// TIA Portal V20 export
FUNCTION_BLOCK "zFNet_10Child"   // FB218, LAD
// stored: MemoryReserve 100, Namespace CITI_Logic, SetENOAutomatically false
   VAR_INPUT
      IN_NumberOf_FN_Retries : Int;   // Number of Timers to Retry the Connection to FNet
      IN_Component_Quantity : Int;   // Number of Child Components
      IN_FN_Response_FLT_Time : DInt;
      IN_OEM_Data : "CITI_Logic.FlexNet_Data";
   END_VAR
   VAR_OUTPUT
      FN_Data : "CITI_Logic.FlexNet_Data";
      FlexNet_White_Light : Bool;
      FlexNet_Green_Light : Bool;
      FlexNet_Buzzer : Bool;
      FlexNet_No_Response_Count : Int;
      FlexNet_DataReceivedByHost : Bool;
      FlexNet_Last_ResponseTime : DInt;
   END_VAR
   VAR
      FN_Dry_Cycle_Block : Bool;
      FN_OneShot : Array[1..32] of Bool;
      Clock_Data : DTL;   // Clock Data used for FlexNet Time Stamp
      System_Time_Tick : Time;   // System Time Tick
      Present_Time_Tick : Int;   // Present Time Tick
      Previous_Time_Tick : Int;   // Previous Time Tick
      Difference_Time_Tick : Int;   // Difference between Present and Previous Tick
      Difference_Time_DInt : DInt;   // Difference in Time
      TimerForFN_DataReady : DInt;   // FlexNet Data Ready Delay
      TimerForFN_Response_Test : DInt;   // FlexNet Response Test
      TimerFN_DataReady_Retry : DInt;   // FlexNet Data Ready Retry Delay
      TimerFN_BuzzerOn : DInt;   // FlexNet No Response Buzzer
      FN_PUNDataRdy_Dly : Bool;   // Start Data Ready Timer
      FN_DataReady_Failed_Retry : Bool;
      FlasherOn : Bool;   // Flasher for StackLights
      FN_NumberOf_Retries : Int;
      FN_Num_Of_Retry_Cnt_HMI : Int;
      FlexNet_Response_FLT_CNT : Int;
      TimerForFlasher : DInt;
      FN_Data_Recd_Delay : Bool;
      Timer_HQ_Delay : DInt;   // FlexNet No Response Buzzer
      Timer_GreenLight_Delay : DInt;   // FlexNet No Response Buzzer
      FN_Num_Of_Retries_CNT : Int;
   END_VAR
   VAR DB_SPECIFIC
      FlexNet_Part_Passed { ExternalAccessible := 'False'; ExternalVisible := 'False'; ExternalWritable := 'False'} : Bool;   // Calculated Part Passed
      FlexNet_Part_Failed { ExternalAccessible := 'False'; ExternalVisible := 'False'; ExternalWritable := 'False'} : Bool;   // Calculated Part Failed
   END_VAR
   VAR
      FlexNet_PassFail_Valid { ExternalAccessible := 'False'; ExternalVisible := 'False'; ExternalWritable := 'False'} : Bool;   // Calculated Valid Part Fail/Pass Data
      ON { ExternalAccessible := 'False'; ExternalVisible := 'False'; ExternalWritable := 'False'} : Bool;   // On
      OFF { ExternalAccessible := 'False'; ExternalVisible := 'False'; ExternalWritable := 'False'} : Bool;   // Off
      ReadClock_Rslt { ExternalAccessible := 'False'; ExternalVisible := 'False'; ExternalWritable := 'False'} : Int;
   END_VAR
   VAR_TEMP   // added for the SCL form of the ladder/FBD networks
      _w1 : Bool;
      _w2 : Bool;
      _w3 : Bool;
      _w4 : Bool;
   END_VAR
BEGIN

REGION Network 1: Always ON and Always OFF Setup
   // Generate local "Always ON" and "Always OFF" conditions
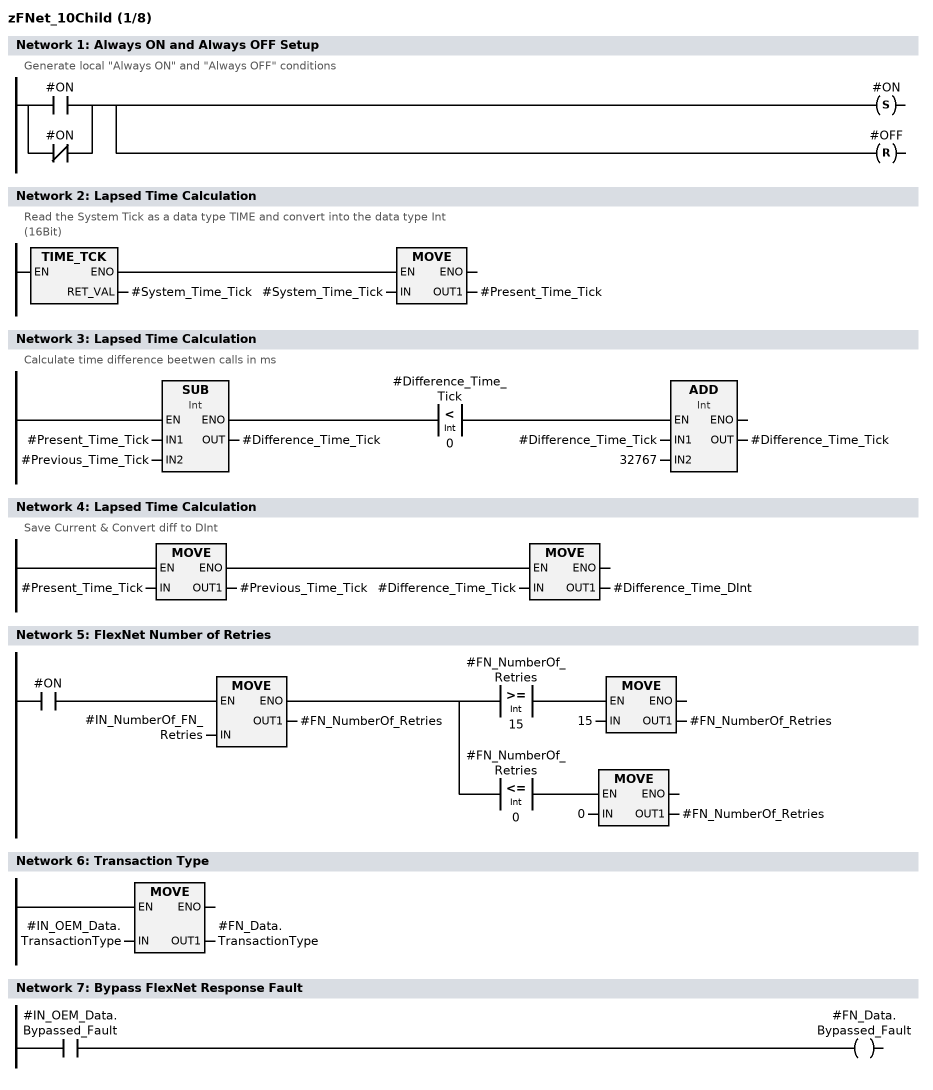
   RUNG wire#powerrail
      Contact( #ON )
      wire#w1
      S_Coil( #ON )
   END_RUNG
   RUNG wire#powerrail
      I_Contact( #ON )
   END_RUNG wire#w1
   RUNG wire#w1
      R_Coil( #OFF )
   END_RUNG
   // the same network as SCL:
   #_w1 := #ON OR NOT #ON;
   IF #_w1 THEN
       #ON := TRUE;
       #OFF := FALSE;
   END_IF;
END_REGION

REGION Network 2: Lapsed Time Calculation
   // Read the System Tick as a data type TIME and convert into the data type Int 
   // (16Bit)
   RUNG wire#powerrail
      TIME_TCK(RET_VAL => #System_Time_Tick)
      { S7_GenerateENO := "TRUE" } Move(in := #System_Time_Tick, out1 => #Present_Time_Tick)
   END_RUNG
   // the same network as SCL:
   #System_Time_Tick := TIME_TCK(ENO => #_w1);
   IF #_w1 THEN #Present_Time_Tick := #System_Time_Tick; END_IF;
END_REGION

REGION Network 3: Lapsed Time Calculation
   // Calculate time difference beetwen calls in ms
   RUNG wire#powerrail
      { S7_Templates := "SrcType := Int"; S7_GenerateENO := "TRUE" } Sub(in1 := #Present_Time_Tick, in2 := #Previous_Time_Tick, out => #Difference_Time_Tick)
      { S7_Templates := "SrcType := Int" } LT_Contact(in1 := #Difference_Time_Tick, in2 := 0)
      { S7_Templates := "SrcType := Int"; S7_GenerateENO := "TRUE" } Add(in1 := #Difference_Time_Tick, in2 := 32767, out => #Difference_Time_Tick)
   END_RUNG
   // the same network as SCL:
   // ENO of a box is taken as its EN; it also drops when the box reports an error
   #Difference_Time_Tick := #Present_Time_Tick - #Previous_Time_Tick;
   IF #Difference_Time_Tick < 0 THEN #Difference_Time_Tick := #Difference_Time_Tick + 32767; END_IF;
END_REGION

REGION Network 4: Lapsed Time Calculation
   // Save Current & Convert diff to DInt
   RUNG wire#powerrail
      { S7_GenerateENO := "TRUE" } Move(in := #Present_Time_Tick, out1 => #Previous_Time_Tick)
      { S7_GenerateENO := "TRUE" } Move(in := #Difference_Time_Tick, out1 => #Difference_Time_DInt)
   END_RUNG
   // the same network as SCL:
   // ENO of a box is taken as its EN; it also drops when the box reports an error
   #Previous_Time_Tick := #Present_Time_Tick;
   #Difference_Time_DInt := #Difference_Time_Tick;
END_REGION

REGION Network 5: FlexNet Number of Retries
   RUNG wire#powerrail
      Contact( #ON )
      { S7_GenerateENO := "TRUE" } Move(in := #IN_NumberOf_FN_Retries, out1 => #FN_NumberOf_Retries)
      wire#w1
      { S7_Templates := "SrcType := Int" } GE_Contact(in1 := #FN_NumberOf_Retries, in2 := 15)
      { S7_GenerateENO := "TRUE" } Move(in := 15, out1 => #FN_NumberOf_Retries)
   END_RUNG
   RUNG wire#w1
      { S7_Templates := "SrcType := Int" } LE_Contact(in1 := #FN_NumberOf_Retries, in2 := 0)
      { S7_GenerateENO := "TRUE" } Move(in := 0, out1 => #FN_NumberOf_Retries)
   END_RUNG
   // the same network as SCL:
   // ENO of a box is taken as its EN; it also drops when the box reports an error
   IF #ON THEN #FN_NumberOf_Retries := #IN_NumberOf_FN_Retries; END_IF;
   IF #ON AND (#FN_NumberOf_Retries >= 15) THEN #FN_NumberOf_Retries := 15; END_IF;
   IF #ON AND (#FN_NumberOf_Retries <= 0) THEN #FN_NumberOf_Retries := 0; END_IF;
END_REGION

REGION Network 6: Transaction Type
   RUNG wire#powerrail
      { S7_GenerateENO := "TRUE" } Move(in := #IN_OEM_Data.TransactionType, out1 => #FN_Data.TransactionType)
   END_RUNG
   // the same network as SCL:
   #FN_Data.TransactionType := #IN_OEM_Data.TransactionType;
END_REGION

REGION Network 7: Bypass FlexNet Response Fault
   RUNG wire#powerrail
      Contact( #IN_OEM_Data.Bypassed_Fault )
      Coil( #FN_Data.Bypassed_Fault )
   END_RUNG
   // the same network as SCL:
   #FN_Data.Bypassed_Fault := #IN_OEM_Data.Bypassed_Fault;
END_REGION

REGION Network 8: Data Reset Input
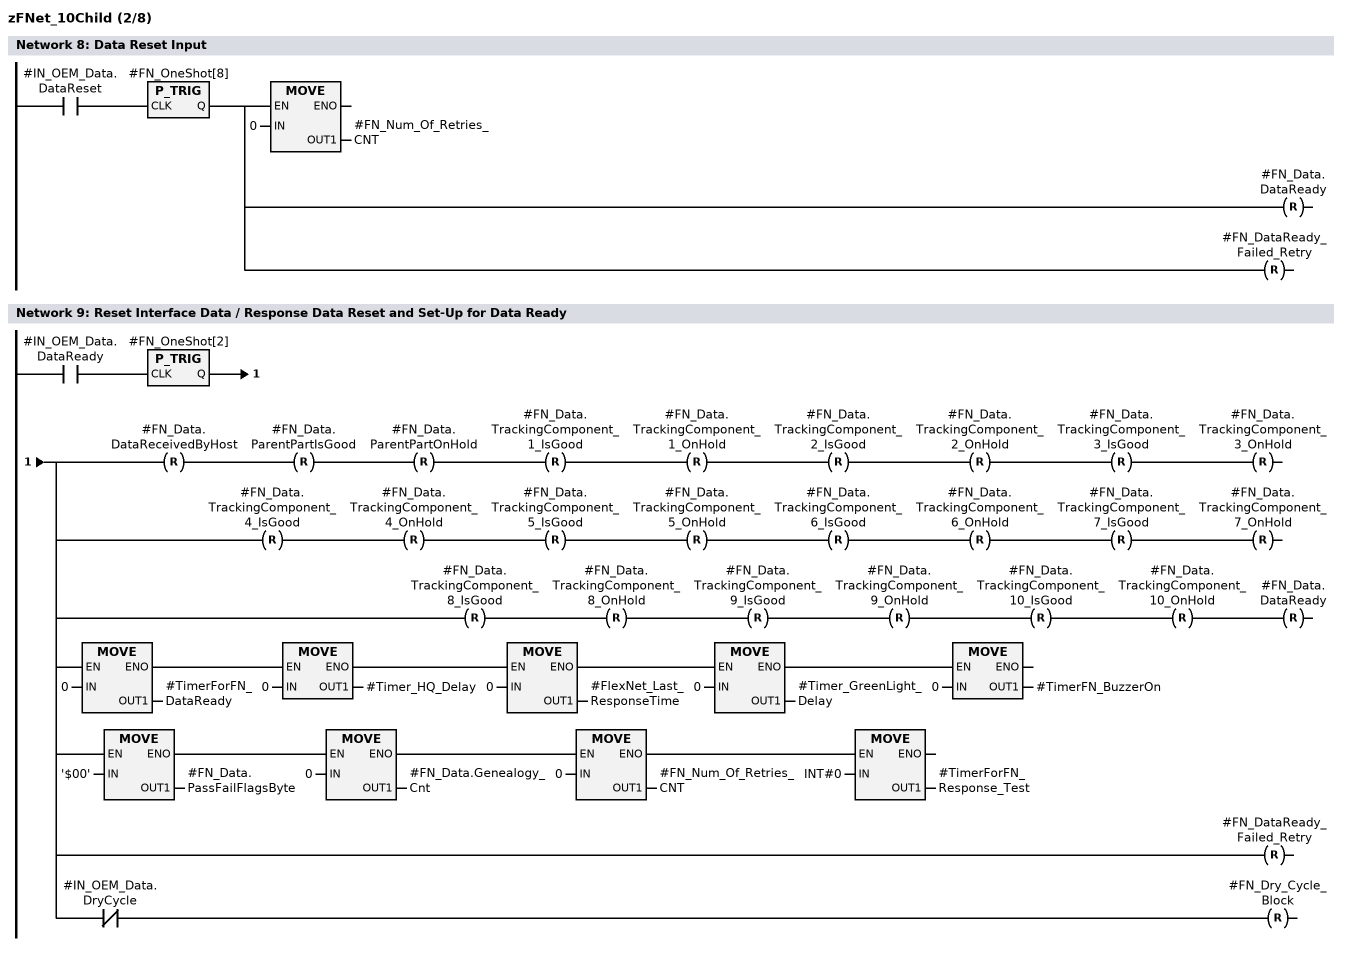
   RUNG wire#powerrail
      Contact( #IN_OEM_Data.DataReset )
      P_Trig( #FN_OneShot[8] )
      wire#w1
      { S7_GenerateENO := "TRUE" } Move(in := 0, out1 => #FN_Num_Of_Retries_CNT)
   END_RUNG
   RUNG wire#w1
      R_Coil( #FN_Data.DataReady )
   END_RUNG
   RUNG wire#w1
      R_Coil( #FN_DataReady_Failed_Retry )
   END_RUNG
   // the same network as SCL:
   #_w1 := #IN_OEM_Data.DataReset AND NOT #FN_OneShot[8];   // rising edge
   #FN_OneShot[8] := #IN_OEM_Data.DataReset;
   IF #_w1 THEN
       #FN_Num_Of_Retries_CNT := 0;
       #FN_Data.DataReady := FALSE;
       #FN_DataReady_Failed_Retry := FALSE;
   END_IF;
END_REGION

REGION Network 9: Reset Interface Data / Response Data Reset and Set-Up for Data Ready
   RUNG wire#powerrail
      Contact( #IN_OEM_Data.DataReady )
      P_Trig( #FN_OneShot[2] )
      wire#w1
      R_Coil( #FN_Data.DataReceivedByHost )
      R_Coil( #FN_Data.ParentPartIsGood )
      R_Coil( #FN_Data.ParentPartOnHold )
      R_Coil( #FN_Data.TrackingComponent_1_IsGood )
      R_Coil( #FN_Data.TrackingComponent_1_OnHold )
      R_Coil( #FN_Data.TrackingComponent_2_IsGood )
      R_Coil( #FN_Data.TrackingComponent_2_OnHold )
      R_Coil( #FN_Data.TrackingComponent_3_IsGood )
      R_Coil( #FN_Data.TrackingComponent_3_OnHold )
   END_RUNG
   RUNG wire#w1
      R_Coil( #FN_Data.TrackingComponent_4_IsGood )
      R_Coil( #FN_Data.TrackingComponent_4_OnHold )
      R_Coil( #FN_Data.TrackingComponent_5_IsGood )
      R_Coil( #FN_Data.TrackingComponent_5_OnHold )
      R_Coil( #FN_Data.TrackingComponent_6_IsGood )
      R_Coil( #FN_Data.TrackingComponent_6_OnHold )
      R_Coil( #FN_Data.TrackingComponent_7_IsGood )
      R_Coil( #FN_Data.TrackingComponent_7_OnHold )
   END_RUNG
   RUNG wire#w1
      R_Coil( #FN_Data.TrackingComponent_8_IsGood )
      R_Coil( #FN_Data.TrackingComponent_8_OnHold )
      R_Coil( #FN_Data.TrackingComponent_9_IsGood )
      R_Coil( #FN_Data.TrackingComponent_9_OnHold )
      R_Coil( #FN_Data.TrackingComponent_10_IsGood )
      R_Coil( #FN_Data.TrackingComponent_10_OnHold )
      R_Coil( #FN_Data.DataReady )
   END_RUNG
   RUNG wire#w1
      Move(in := 0, out1 => #TimerForFN_DataReady)
      Move(in := 0, out1 => #Timer_HQ_Delay)
      Move(in := 0, out1 => #FlexNet_Last_ResponseTime)
      Move(in := 0, out1 => #Timer_GreenLight_Delay)
      { S7_GenerateENO := "TRUE" } Move(in := 0, out1 => #TimerFN_BuzzerOn)
   END_RUNG
   RUNG wire#w1
      { S7_GenerateENO := "TRUE" } Move(in := '$00', out1 => #FN_Data.PassFailFlagsByte)
      Move(in := 0, out1 => #FN_Data.Genealogy_Cnt)
      { S7_GenerateENO := "TRUE" } Move(in := 0, out1 => #FN_Num_Of_Retries_CNT)
      { S7_GenerateENO := "TRUE" } Move(in := INT#0, out1 => #TimerForFN_Response_Test)
   END_RUNG
   RUNG wire#w1
      R_Coil( #FN_DataReady_Failed_Retry )
   END_RUNG
   RUNG wire#w1
      I_Contact( #IN_OEM_Data.DryCycle )
      R_Coil( #FN_Dry_Cycle_Block )
   END_RUNG
   // the same network as SCL:
   // ENO of a box is taken as its EN; it also drops when the box reports an error
   #_w1 := #IN_OEM_Data.DataReady AND NOT #FN_OneShot[2];   // rising edge
   #FN_OneShot[2] := #IN_OEM_Data.DataReady;
   IF #_w1 THEN
       #FN_Data.DataReceivedByHost := FALSE;
       #FN_Data.ParentPartIsGood := FALSE;
       #FN_Data.ParentPartOnHold := FALSE;
       #FN_Data.TrackingComponent_1_IsGood := FALSE;
       #FN_Data.TrackingComponent_1_OnHold := FALSE;
       #FN_Data.TrackingComponent_2_IsGood := FALSE;
       #FN_Data.TrackingComponent_2_OnHold := FALSE;
       #FN_Data.TrackingComponent_3_IsGood := FALSE;
       #FN_Data.TrackingComponent_3_OnHold := FALSE;
       #FN_Data.TrackingComponent_4_IsGood := FALSE;
       #FN_Data.TrackingComponent_4_OnHold := FALSE;
       #FN_Data.TrackingComponent_5_IsGood := FALSE;
       #FN_Data.TrackingComponent_5_OnHold := FALSE;
       #FN_Data.TrackingComponent_6_IsGood := FALSE;
       #FN_Data.TrackingComponent_6_OnHold := FALSE;
       #FN_Data.TrackingComponent_7_IsGood := FALSE;
       #FN_Data.TrackingComponent_7_OnHold := FALSE;
       #FN_Data.TrackingComponent_8_IsGood := FALSE;
       #FN_Data.TrackingComponent_8_OnHold := FALSE;
       #FN_Data.TrackingComponent_9_IsGood := FALSE;
       #FN_Data.TrackingComponent_9_OnHold := FALSE;
       #FN_Data.TrackingComponent_10_IsGood := FALSE;
       #FN_Data.TrackingComponent_10_OnHold := FALSE;
       #FN_Data.DataReady := FALSE;
       #TimerForFN_DataReady := 0;
       #Timer_HQ_Delay := 0;
       #FlexNet_Last_ResponseTime := 0;
       #Timer_GreenLight_Delay := 0;
       #TimerFN_BuzzerOn := 0;
       #FN_Data.PassFailFlagsByte := '$00';
       #FN_Data.Genealogy_Cnt := 0;
       #FN_Num_Of_Retries_CNT := 0;
       #TimerForFN_Response_Test := INT#0;
       #FN_DataReady_Failed_Retry := FALSE;
   END_IF;
   IF #_w1 AND NOT #IN_OEM_Data.DryCycle THEN #FN_Dry_Cycle_Block := FALSE; END_IF;
END_REGION

REGION Network 10: Test Part Failed or Passed signals Using the Transaction Byte to enable certain test parameters
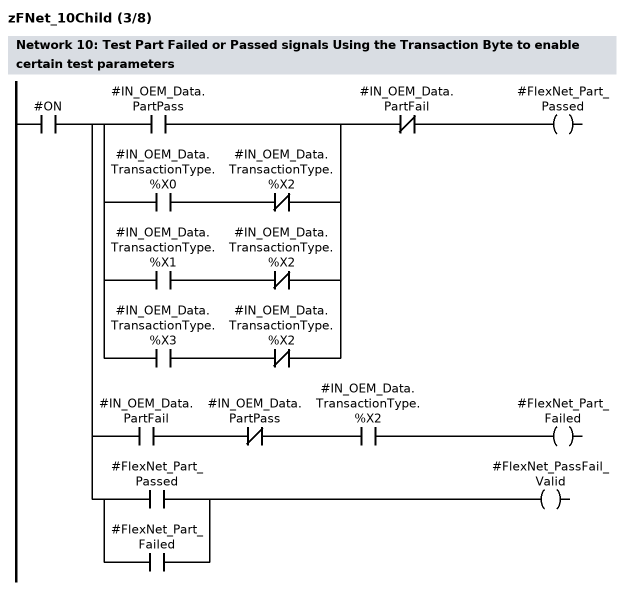
   RUNG wire#powerrail
      Contact( #ON )
      wire#w1
      Contact( #IN_OEM_Data.PartPass )
      wire#w2
      I_Contact( #IN_OEM_Data.PartFail )
      Coil( #FlexNet_Part_Passed )
   END_RUNG
   RUNG wire#w1
      Contact( #IN_OEM_Data.TransactionType.%X0 )
      I_Contact( #IN_OEM_Data.TransactionType.%X2 )
   END_RUNG wire#w2
   RUNG wire#w1
      Contact( #IN_OEM_Data.TransactionType.%X1 )
      I_Contact( #IN_OEM_Data.TransactionType.%X2 )
   END_RUNG wire#w2
   RUNG wire#w1
      Contact( #IN_OEM_Data.TransactionType.%X3 )
      I_Contact( #IN_OEM_Data.TransactionType.%X2 )
   END_RUNG wire#w2
   RUNG wire#w1
      Contact( #IN_OEM_Data.PartFail )
      I_Contact( #IN_OEM_Data.PartPass )
      Contact( #IN_OEM_Data.TransactionType.%X2 )
      Coil( #FlexNet_Part_Failed )
   END_RUNG
   RUNG wire#w1
      Contact( #FlexNet_Part_Passed )
      wire#w3
      Coil( #FlexNet_PassFail_Valid )
   END_RUNG
   RUNG wire#w1
      Contact( #FlexNet_Part_Failed )
   END_RUNG wire#w3
   // the same network as SCL:
   #FlexNet_Part_Passed := #ON AND (#IN_OEM_Data.PartPass OR (#IN_OEM_Data.TransactionType.%X0 AND NOT #IN_OEM_Data.TransactionType.%X2) OR (#IN_OEM_Data.TransactionType.%X1 AND NOT #IN_OEM_Data.TransactionType.%X2) OR (#IN_OEM_Data.TransactionType.%X3 AND NOT #IN_OEM_Data.TransactionType.%X2)) AND NOT #IN_OEM_Data.PartFail;
   #FlexNet_Part_Failed := #ON AND #IN_OEM_Data.PartFail AND NOT #IN_OEM_Data.PartPass AND #IN_OEM_Data.TransactionType.%X2;
   #FlexNet_PassFail_Valid := #ON AND (#FlexNet_Part_Passed OR #FlexNet_Part_Failed);
END_REGION

REGION Network 11: Copy PUN Data, Tracking ID/Attribute, Clock Data, Part Pass/Fail Data into FlexNet Registers
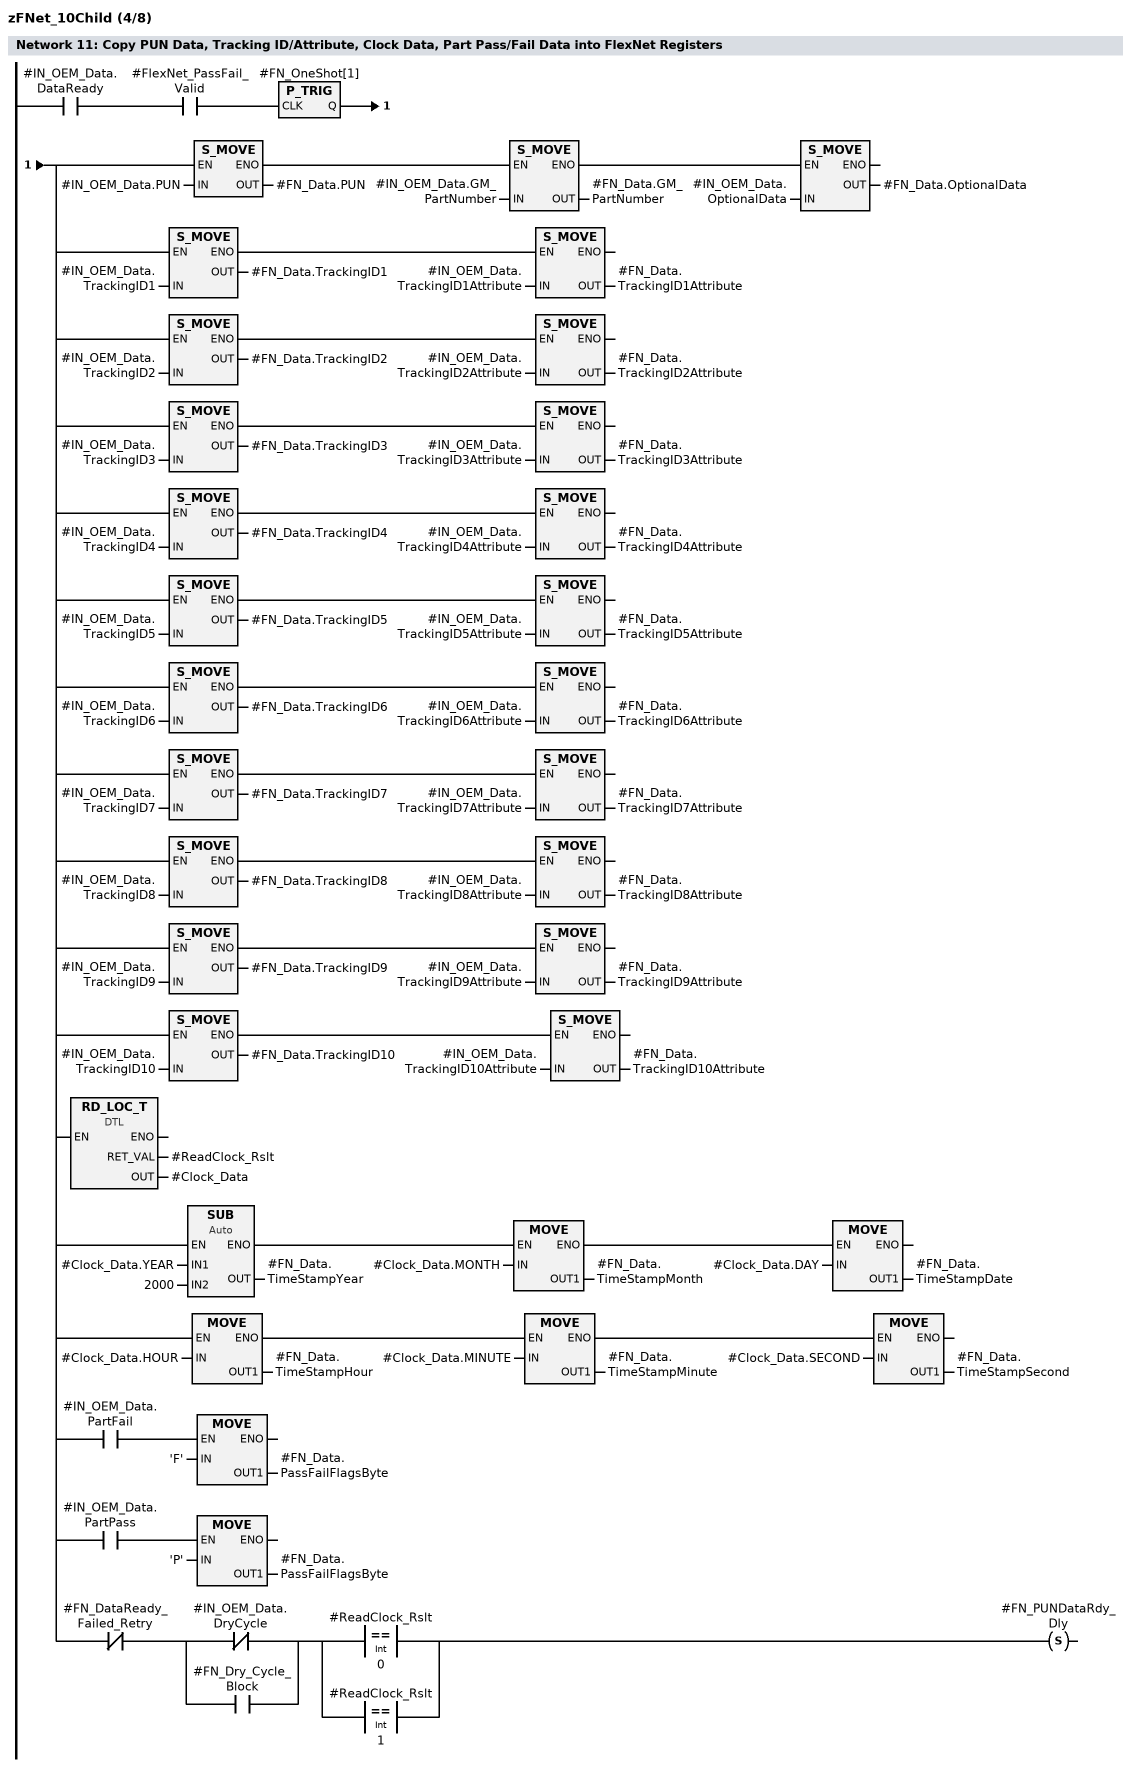
   RUNG wire#powerrail
      Contact( #IN_OEM_Data.DataReady )
      Contact( #FlexNet_PassFail_Valid )
      P_Trig( #FN_OneShot[1] )
      wire#w1
      S_Move(in := #IN_OEM_Data.PUN, out => #FN_Data.PUN)
      S_Move(in := #IN_OEM_Data.GM_PartNumber, out => #FN_Data.GM_PartNumber)
      S_Move(in := #IN_OEM_Data.OptionalData, out => #FN_Data.OptionalData)
   END_RUNG
   RUNG wire#w1
      S_Move(in := #IN_OEM_Data.TrackingID1, out => #FN_Data.TrackingID1)
      S_Move(in := #IN_OEM_Data.TrackingID1Attribute, out => #FN_Data.TrackingID1Attribute)
   END_RUNG
   RUNG wire#w1
      S_Move(in := #IN_OEM_Data.TrackingID2, out => #FN_Data.TrackingID2)
      S_Move(in := #IN_OEM_Data.TrackingID2Attribute, out => #FN_Data.TrackingID2Attribute)
   END_RUNG
   RUNG wire#w1
      S_Move(in := #IN_OEM_Data.TrackingID3, out => #FN_Data.TrackingID3)
      S_Move(in := #IN_OEM_Data.TrackingID3Attribute, out => #FN_Data.TrackingID3Attribute)
   END_RUNG
   RUNG wire#w1
      S_Move(in := #IN_OEM_Data.TrackingID4, out => #FN_Data.TrackingID4)
      S_Move(in := #IN_OEM_Data.TrackingID4Attribute, out => #FN_Data.TrackingID4Attribute)
   END_RUNG
   RUNG wire#w1
      S_Move(in := #IN_OEM_Data.TrackingID5, out => #FN_Data.TrackingID5)
      S_Move(in := #IN_OEM_Data.TrackingID5Attribute, out => #FN_Data.TrackingID5Attribute)
   END_RUNG
   RUNG wire#w1
      S_Move(in := #IN_OEM_Data.TrackingID6, out => #FN_Data.TrackingID6)
      S_Move(in := #IN_OEM_Data.TrackingID6Attribute, out => #FN_Data.TrackingID6Attribute)
   END_RUNG
   RUNG wire#w1
      S_Move(in := #IN_OEM_Data.TrackingID7, out => #FN_Data.TrackingID7)
      S_Move(in := #IN_OEM_Data.TrackingID7Attribute, out => #FN_Data.TrackingID7Attribute)
   END_RUNG
   RUNG wire#w1
      S_Move(in := #IN_OEM_Data.TrackingID8, out => #FN_Data.TrackingID8)
      S_Move(in := #IN_OEM_Data.TrackingID8Attribute, out => #FN_Data.TrackingID8Attribute)
   END_RUNG
   RUNG wire#w1
      S_Move(in := #IN_OEM_Data.TrackingID9, out => #FN_Data.TrackingID9)
      S_Move(in := #IN_OEM_Data.TrackingID9Attribute, out => #FN_Data.TrackingID9Attribute)
   END_RUNG
   RUNG wire#w1
      S_Move(in := #IN_OEM_Data.TrackingID10, out => #FN_Data.TrackingID10)
      S_Move(in := #IN_OEM_Data.TrackingID10Attribute, out => #FN_Data.TrackingID10Attribute)
   END_RUNG
   RUNG wire#w1
      { S7_Templates := "date_type := DTL" } RD_LOC_T(RET_VAL => #ReadClock_Rslt, OUT => #Clock_Data)
   END_RUNG
   RUNG wire#w1
      Sub(in1 := #Clock_Data.YEAR, in2 := 2000, out => #FN_Data.TimeStampYear)
      Move(in := #Clock_Data.MONTH, out1 => #FN_Data.TimeStampMonth)
      Move(in := #Clock_Data.DAY, out1 => #FN_Data.TimeStampDate)
   END_RUNG
   RUNG wire#w1
      Move(in := #Clock_Data.HOUR, out1 => #FN_Data.TimeStampHour)
      Move(in := #Clock_Data.MINUTE, out1 => #FN_Data.TimeStampMinute)
      Move(in := #Clock_Data.SECOND, out1 => #FN_Data.TimeStampSecond)
   END_RUNG
   RUNG wire#w1
      Contact( #IN_OEM_Data.PartFail )
      Move(in := 'F', out1 => #FN_Data.PassFailFlagsByte)
   END_RUNG
   RUNG wire#w1
      Contact( #IN_OEM_Data.PartPass )
      Move(in := 'P', out1 => #FN_Data.PassFailFlagsByte)
   END_RUNG
   RUNG wire#w1
      I_Contact( #FN_DataReady_Failed_Retry )
      wire#w2
      I_Contact( #IN_OEM_Data.DryCycle )
      wire#w3
      { S7_Templates := "SrcType := Int" } EQ_Contact(in1 := #ReadClock_Rslt, in2 := 0)
      wire#w4
      S_Coil( #FN_PUNDataRdy_Dly )
   END_RUNG
   RUNG wire#w2
      Contact( #FN_Dry_Cycle_Block )
   END_RUNG wire#w3
   RUNG wire#w3
      { S7_Templates := "SrcType := Int" } EQ_Contact(in1 := #ReadClock_Rslt, in2 := 1)
   END_RUNG wire#w4
   // the same network as SCL:
   #_w1 := #IN_OEM_Data.DataReady AND #FlexNet_PassFail_Valid;
   #_w2 := #_w1 AND NOT #FN_OneShot[1];   // rising edge
   #FN_OneShot[1] := #_w1;
   IF #_w2 THEN
       #FN_Data.PUN := #IN_OEM_Data.PUN;
       #FN_Data.GM_PartNumber := #IN_OEM_Data.GM_PartNumber;
       #FN_Data.OptionalData := #IN_OEM_Data.OptionalData;
       #FN_Data.TrackingID1 := #IN_OEM_Data.TrackingID1;
       #FN_Data.TrackingID1Attribute := #IN_OEM_Data.TrackingID1Attribute;
       #FN_Data.TrackingID2 := #IN_OEM_Data.TrackingID2;
       #FN_Data.TrackingID2Attribute := #IN_OEM_Data.TrackingID2Attribute;
       #FN_Data.TrackingID3 := #IN_OEM_Data.TrackingID3;
       #FN_Data.TrackingID3Attribute := #IN_OEM_Data.TrackingID3Attribute;
       #FN_Data.TrackingID4 := #IN_OEM_Data.TrackingID4;
       #FN_Data.TrackingID4Attribute := #IN_OEM_Data.TrackingID4Attribute;
       #FN_Data.TrackingID5 := #IN_OEM_Data.TrackingID5;
       #FN_Data.TrackingID5Attribute := #IN_OEM_Data.TrackingID5Attribute;
       #FN_Data.TrackingID6 := #IN_OEM_Data.TrackingID6;
       #FN_Data.TrackingID6Attribute := #IN_OEM_Data.TrackingID6Attribute;
       #FN_Data.TrackingID7 := #IN_OEM_Data.TrackingID7;
       #FN_Data.TrackingID7Attribute := #IN_OEM_Data.TrackingID7Attribute;
       #FN_Data.TrackingID8 := #IN_OEM_Data.TrackingID8;
       #FN_Data.TrackingID8Attribute := #IN_OEM_Data.TrackingID8Attribute;
       #FN_Data.TrackingID9 := #IN_OEM_Data.TrackingID9;
       #FN_Data.TrackingID9Attribute := #IN_OEM_Data.TrackingID9Attribute;
       #FN_Data.TrackingID10 := #IN_OEM_Data.TrackingID10;
       #FN_Data.TrackingID10Attribute := #IN_OEM_Data.TrackingID10Attribute;
       #ReadClock_Rslt := RD_LOC_T(OUT => #Clock_Data);
       #FN_Data.TimeStampYear := #Clock_Data.YEAR - 2000;
       #FN_Data.TimeStampMonth := #Clock_Data.MONTH;
       #FN_Data.TimeStampDate := #Clock_Data.DAY;
       #FN_Data.TimeStampHour := #Clock_Data.HOUR;
       #FN_Data.TimeStampMinute := #Clock_Data.MINUTE;
       #FN_Data.TimeStampSecond := #Clock_Data.SECOND;
   END_IF;
   IF #_w2 AND #IN_OEM_Data.PartFail THEN #FN_Data.PassFailFlagsByte := 'F'; END_IF;
   IF #_w2 AND #IN_OEM_Data.PartPass THEN #FN_Data.PassFailFlagsByte := 'P'; END_IF;
   IF #_w2 AND NOT #FN_DataReady_Failed_Retry AND (NOT #IN_OEM_Data.DryCycle OR #FN_Dry_Cycle_Block) AND ((#ReadClock_Rslt = 0) OR (#ReadClock_Rslt = 1)) THEN
       #FN_PUNDataRdy_Dly := TRUE;
   END_IF;
END_REGION

REGION Network 12: Turn On FlexNet DataReady. Reset PUN Data Ready Delay and Failed Retry Data Ready
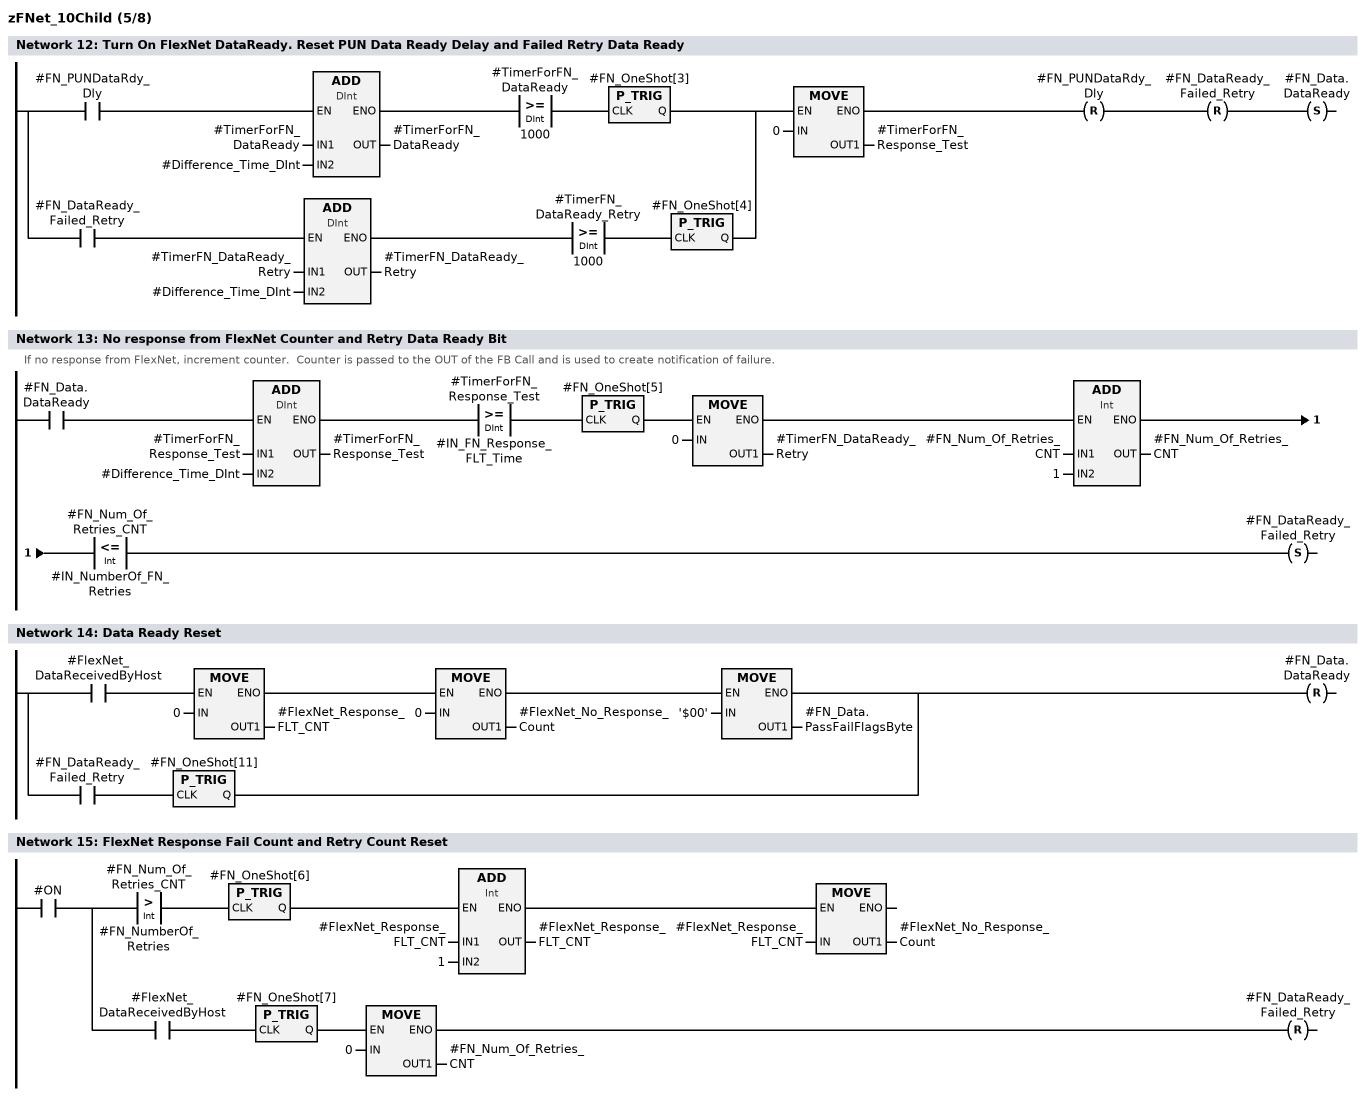
   RUNG wire#powerrail
      Contact( #FN_PUNDataRdy_Dly )
      { S7_Templates := "SrcType := DInt"; S7_GenerateENO := "TRUE" } Add(in1 := #TimerForFN_DataReady, in2 := #Difference_Time_DInt, out => #TimerForFN_DataReady)
      { S7_Templates := "SrcType := DInt" } GE_Contact(in1 := #TimerForFN_DataReady, in2 := 1000)
      P_Trig( #FN_OneShot[3] )
      wire#w1
      { S7_GenerateENO := "TRUE" } Move(in := 0, out1 => #TimerForFN_Response_Test)
      R_Coil( #FN_PUNDataRdy_Dly )
      R_Coil( #FN_DataReady_Failed_Retry )
      S_Coil( #FN_Data.DataReady )
   END_RUNG
   RUNG wire#powerrail
      Contact( #FN_DataReady_Failed_Retry )
      { S7_Templates := "SrcType := DInt"; S7_GenerateENO := "TRUE" } Add(in1 := #TimerFN_DataReady_Retry, in2 := #Difference_Time_DInt, out => #TimerFN_DataReady_Retry)
      { S7_Templates := "SrcType := DInt" } GE_Contact(in1 := #TimerFN_DataReady_Retry, in2 := 1000)
      P_Trig( #FN_OneShot[4] )
   END_RUNG wire#w1
   // the same network as SCL:
   // ENO of a box is taken as its EN; it also drops when the box reports an error
   IF #FN_PUNDataRdy_Dly THEN #TimerForFN_DataReady := #TimerForFN_DataReady + #Difference_Time_DInt; END_IF;
   #_w1 := #FN_PUNDataRdy_Dly AND (#TimerForFN_DataReady >= 1000);
   #_w2 := #_w1 AND NOT #FN_OneShot[3];   // rising edge
   #FN_OneShot[3] := #_w1;
   IF #FN_DataReady_Failed_Retry THEN
       #TimerFN_DataReady_Retry := #TimerFN_DataReady_Retry + #Difference_Time_DInt;
   END_IF;
   #_w3 := #FN_DataReady_Failed_Retry AND (#TimerFN_DataReady_Retry >= 1000);
   #_w4 := #_w3 AND NOT #FN_OneShot[4];   // rising edge
   #FN_OneShot[4] := #_w3;
   IF #_w2 OR #_w4 THEN
       #TimerForFN_Response_Test := 0;
       #FN_PUNDataRdy_Dly := FALSE;
       #FN_DataReady_Failed_Retry := FALSE;
       #FN_Data.DataReady := TRUE;
   END_IF;
END_REGION

REGION Network 13: No response from FlexNet Counter and Retry Data Ready Bit
   // If no response from FlexNet, increment counter.  Counter is passed to the OUT of the FB Call and is used to create notification of failure.
   RUNG wire#powerrail
      Contact( #FN_Data.DataReady )
      { S7_Templates := "SrcType := DInt"; S7_GenerateENO := "TRUE" } Add(in1 := #TimerForFN_Response_Test, in2 := #Difference_Time_DInt, out => #TimerForFN_Response_Test)
      { S7_Templates := "SrcType := DInt" } GE_Contact(in1 := #TimerForFN_Response_Test, in2 := #IN_FN_Response_FLT_Time)
      P_Trig( #FN_OneShot[5] )
      { S7_GenerateENO := "TRUE" } Move(in := 0, out1 => #TimerFN_DataReady_Retry)
      { S7_Templates := "SrcType := Int"; S7_GenerateENO := "TRUE" } Add(in1 := #FN_Num_Of_Retries_CNT, in2 := 1, out => #FN_Num_Of_Retries_CNT)
      { S7_Templates := "SrcType := Int" } LE_Contact(in1 := #FN_Num_Of_Retries_CNT, in2 := #IN_NumberOf_FN_Retries)
      S_Coil( #FN_DataReady_Failed_Retry )
   END_RUNG
   // the same network as SCL:
   // ENO of a box is taken as its EN; it also drops when the box reports an error
   IF #FN_Data.DataReady THEN
       #TimerForFN_Response_Test := #TimerForFN_Response_Test + #Difference_Time_DInt;
   END_IF;
   #_w1 := #FN_Data.DataReady AND (#TimerForFN_Response_Test >= #IN_FN_Response_FLT_Time);
   #_w2 := #_w1 AND NOT #FN_OneShot[5];   // rising edge
   #FN_OneShot[5] := #_w1;
   IF #_w2 THEN
       #TimerFN_DataReady_Retry := 0;
       #FN_Num_Of_Retries_CNT := #FN_Num_Of_Retries_CNT + 1;
   END_IF;
   IF #_w2 AND (#FN_Num_Of_Retries_CNT <= #IN_NumberOf_FN_Retries) THEN
       #FN_DataReady_Failed_Retry := TRUE;
   END_IF;
END_REGION

REGION Network 14: Data Ready Reset
   RUNG wire#powerrail
      Contact( #FlexNet_DataReceivedByHost )
      { S7_GenerateENO := "TRUE" } Move(in := 0, out1 => #FlexNet_Response_FLT_CNT)
      { S7_GenerateENO := "TRUE" } Move(in := 0, out1 => #FlexNet_No_Response_Count)
      { S7_GenerateENO := "TRUE" } Move(in := '$00', out1 => #FN_Data.PassFailFlagsByte)
      wire#w1
      R_Coil( #FN_Data.DataReady )
   END_RUNG
   RUNG wire#powerrail
      Contact( #FN_DataReady_Failed_Retry )
      P_Trig( #FN_OneShot[11] )
   END_RUNG wire#w1
   // the same network as SCL:
   // ENO of a box is taken as its EN; it also drops when the box reports an error
   IF #FlexNet_DataReceivedByHost THEN
       #FlexNet_Response_FLT_CNT := 0;
       #FlexNet_No_Response_Count := 0;
       #FN_Data.PassFailFlagsByte := '$00';
   END_IF;
   #_w1 := #FN_DataReady_Failed_Retry AND NOT #FN_OneShot[11];   // rising edge
   #FN_OneShot[11] := #FN_DataReady_Failed_Retry;
   IF #FlexNet_DataReceivedByHost OR #_w1 THEN #FN_Data.DataReady := FALSE; END_IF;
END_REGION

REGION Network 15: FlexNet Response Fail Count and Retry Count Reset
   RUNG wire#powerrail
      Contact( #ON )
      wire#w1
      { S7_Templates := "SrcType := Int" } GT_Contact(in1 := #FN_Num_Of_Retries_CNT, in2 := #FN_NumberOf_Retries)
      P_Trig( #FN_OneShot[6] )
      { S7_Templates := "SrcType := Int"; S7_GenerateENO := "TRUE" } Add(in1 := #FlexNet_Response_FLT_CNT, in2 := 1, out => #FlexNet_Response_FLT_CNT)
      { S7_GenerateENO := "TRUE" } Move(in := #FlexNet_Response_FLT_CNT, out1 => #FlexNet_No_Response_Count)
   END_RUNG
   RUNG wire#w1
      Contact( #FlexNet_DataReceivedByHost )
      P_Trig( #FN_OneShot[7] )
      { S7_GenerateENO := "TRUE" } Move(in := 0, out1 => #FN_Num_Of_Retries_CNT)
      R_Coil( #FN_DataReady_Failed_Retry )
   END_RUNG
   // the same network as SCL:
   // ENO of a box is taken as its EN; it also drops when the box reports an error
   #_w1 := #ON AND (#FN_Num_Of_Retries_CNT > #FN_NumberOf_Retries);
   #_w2 := #_w1 AND NOT #FN_OneShot[6];   // rising edge
   #FN_OneShot[6] := #_w1;
   IF #_w2 THEN
       #FlexNet_Response_FLT_CNT := #FlexNet_Response_FLT_CNT + 1;
       #FlexNet_No_Response_Count := #FlexNet_Response_FLT_CNT;
   END_IF;
   #_w3 := #ON AND #FlexNet_DataReceivedByHost;
   #_w4 := #_w3 AND NOT #FN_OneShot[7];   // rising edge
   #FN_OneShot[7] := #_w3;
   IF #_w4 THEN
       #FN_Num_Of_Retries_CNT := 0;
       #FN_DataReady_Failed_Retry := FALSE;
   END_IF;
END_REGION

REGION Network 16: Data Received By Host Output and Delay for HQ to Wait for Server Response
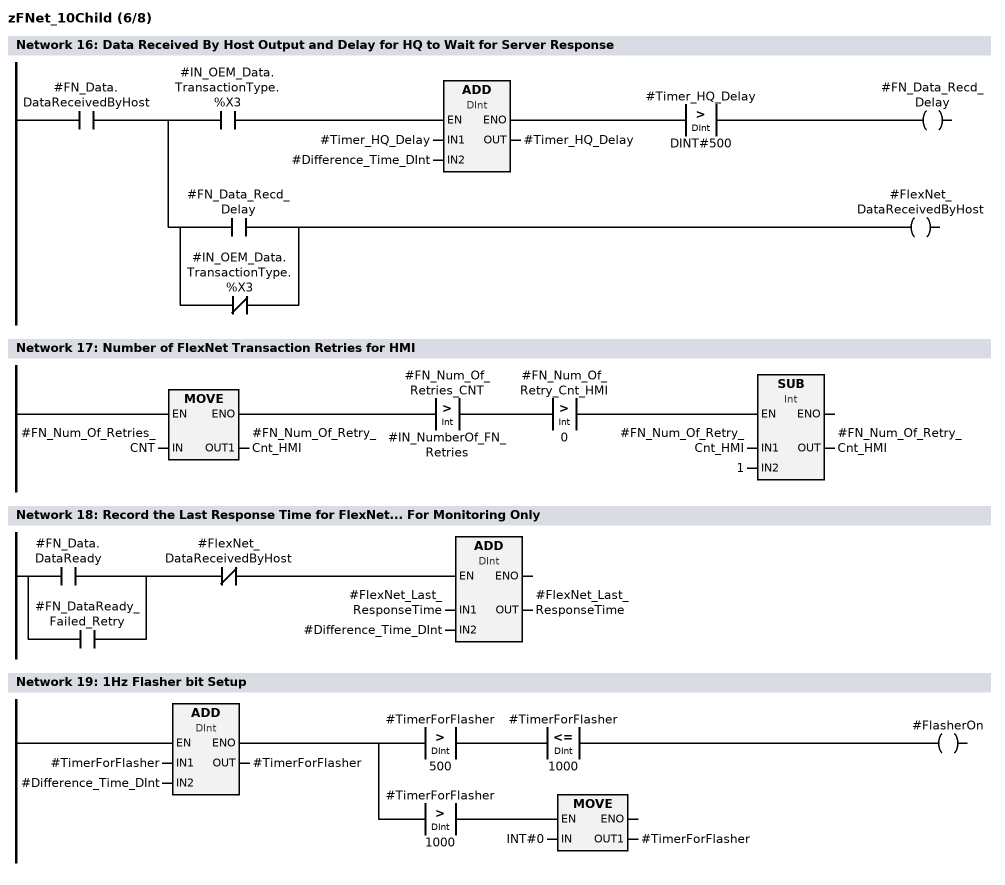
   RUNG wire#powerrail
      Contact( #FN_Data.DataReceivedByHost )
      wire#w1
      Contact( #IN_OEM_Data.TransactionType.%X3 )
      { S7_Templates := "SrcType := DInt" } Add(in1 := #Timer_HQ_Delay, in2 := #Difference_Time_DInt, out => #Timer_HQ_Delay)
      { S7_Templates := "SrcType := DInt" } GT_Contact(in1 := #Timer_HQ_Delay, in2 := DINT#500)
      Coil( #FN_Data_Recd_Delay )
   END_RUNG
   RUNG wire#w1
      Contact( #FN_Data_Recd_Delay )
      wire#w2
      Coil( #FlexNet_DataReceivedByHost )
   END_RUNG
   RUNG wire#w1
      I_Contact( #IN_OEM_Data.TransactionType.%X3 )
   END_RUNG wire#w2
   // the same network as SCL:
   #_w1 := #FN_Data.DataReceivedByHost AND #IN_OEM_Data.TransactionType.%X3;
   IF #_w1 THEN #Timer_HQ_Delay := #Timer_HQ_Delay + #Difference_Time_DInt; END_IF;
   #FN_Data_Recd_Delay := #_w1 AND (#Timer_HQ_Delay > DINT#500);
   #FlexNet_DataReceivedByHost := #FN_Data.DataReceivedByHost AND (#FN_Data_Recd_Delay OR NOT #IN_OEM_Data.TransactionType.%X3);
END_REGION

REGION Network 17: Number of FlexNet Transaction Retries for HMI
   RUNG wire#powerrail
      { S7_GenerateENO := "TRUE" } Move(in := #FN_Num_Of_Retries_CNT, out1 => #FN_Num_Of_Retry_Cnt_HMI)
      { S7_Templates := "SrcType := Int" } GT_Contact(in1 := #FN_Num_Of_Retries_CNT, in2 := #IN_NumberOf_FN_Retries)
      { S7_Templates := "SrcType := Int" } GT_Contact(in1 := #FN_Num_Of_Retry_Cnt_HMI, in2 := 0)
      { S7_Templates := "SrcType := Int"; S7_GenerateENO := "TRUE" } Sub(in1 := #FN_Num_Of_Retry_Cnt_HMI, in2 := 1, out => #FN_Num_Of_Retry_Cnt_HMI)
   END_RUNG
   // the same network as SCL:
   // ENO of a box is taken as its EN; it also drops when the box reports an error
   #FN_Num_Of_Retry_Cnt_HMI := #FN_Num_Of_Retries_CNT;
   IF (#FN_Num_Of_Retries_CNT > #IN_NumberOf_FN_Retries) AND (#FN_Num_Of_Retry_Cnt_HMI > 0) THEN
       #FN_Num_Of_Retry_Cnt_HMI := #FN_Num_Of_Retry_Cnt_HMI - 1;
   END_IF;
END_REGION

REGION Network 18: Record the Last Response Time for FlexNet... For Monitoring Only
   RUNG wire#powerrail
      Contact( #FN_Data.DataReady )
      wire#w1
      I_Contact( #FlexNet_DataReceivedByHost )
      { S7_Templates := "SrcType := DInt"; S7_GenerateENO := "TRUE" } Add(in1 := #FlexNet_Last_ResponseTime, in2 := #Difference_Time_DInt, out => #FlexNet_Last_ResponseTime)
   END_RUNG
   RUNG wire#powerrail
      Contact( #FN_DataReady_Failed_Retry )
   END_RUNG wire#w1
   // the same network as SCL:
   IF (#FN_Data.DataReady OR #FN_DataReady_Failed_Retry) AND NOT #FlexNet_DataReceivedByHost THEN
       #FlexNet_Last_ResponseTime := #FlexNet_Last_ResponseTime + #Difference_Time_DInt;
   END_IF;
END_REGION

REGION Network 19: 1Hz Flasher bit Setup
   RUNG wire#powerrail
      { S7_Templates := "SrcType := DInt"; S7_GenerateENO := "TRUE" } Add(in1 := #TimerForFlasher, in2 := #Difference_Time_DInt, out => #TimerForFlasher)
      wire#w1
      { S7_Templates := "SrcType := DInt" } GT_Contact(in1 := #TimerForFlasher, in2 := 500)
      { S7_Templates := "SrcType := DInt" } LE_Contact(in1 := #TimerForFlasher, in2 := 1000)
      Coil( #FlasherOn )
   END_RUNG
   RUNG wire#w1
      { S7_Templates := "SrcType := DInt" } GT_Contact(in1 := #TimerForFlasher, in2 := 1000)
      { S7_GenerateENO := "TRUE" } Move(in := INT#0, out1 => #TimerForFlasher)
   END_RUNG
   // the same network as SCL:
   // ENO of a box is taken as its EN; it also drops when the box reports an error
   #TimerForFlasher := #TimerForFlasher + #Difference_Time_DInt;
   #FlasherOn := (#TimerForFlasher > 500) AND (#TimerForFlasher <= 1000);
   IF #TimerForFlasher > 1000 THEN #TimerForFlasher := INT#0; END_IF;
END_REGION

REGION Network 20: White Light Flashing
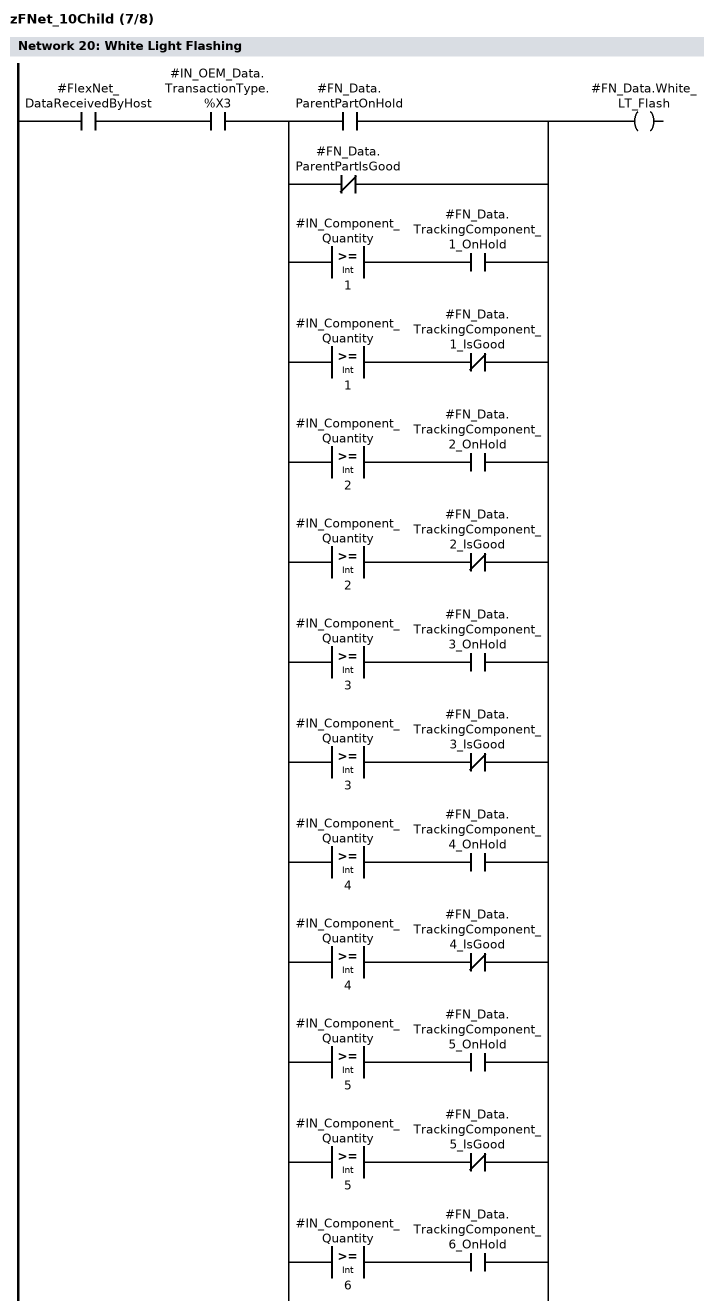
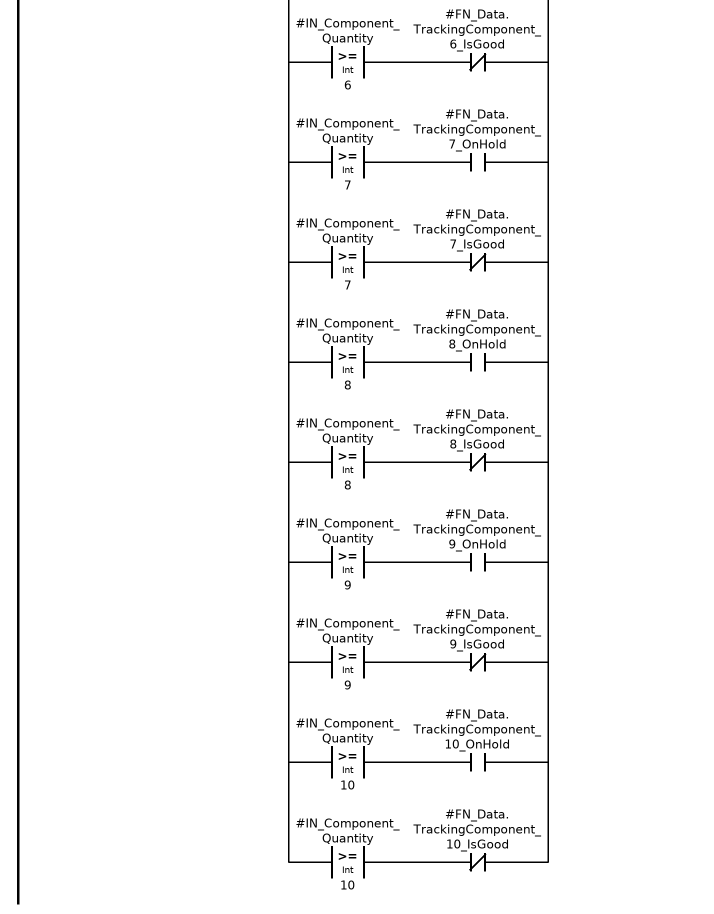
   RUNG wire#powerrail
      Contact( #FlexNet_DataReceivedByHost )
      Contact( #IN_OEM_Data.TransactionType.%X3 )
      wire#w1
      Contact( #FN_Data.ParentPartOnHold )
      wire#w2
      Coil( #FN_Data.White_LT_Flash )
   END_RUNG
   RUNG wire#w1
      I_Contact( #FN_Data.ParentPartIsGood )
   END_RUNG wire#w2
   RUNG wire#w1
      { S7_Templates := "SrcType := Int" } GE_Contact(in1 := #IN_Component_Quantity, in2 := 1)
      Contact( #FN_Data.TrackingComponent_1_OnHold )
   END_RUNG wire#w2
   RUNG wire#w1
      { S7_Templates := "SrcType := Int" } GE_Contact(in1 := #IN_Component_Quantity, in2 := 1)
      I_Contact( #FN_Data.TrackingComponent_1_IsGood )
   END_RUNG wire#w2
   RUNG wire#w1
      { S7_Templates := "SrcType := Int" } GE_Contact(in1 := #IN_Component_Quantity, in2 := 2)
      Contact( #FN_Data.TrackingComponent_2_OnHold )
   END_RUNG wire#w2
   RUNG wire#w1
      { S7_Templates := "SrcType := Int" } GE_Contact(in1 := #IN_Component_Quantity, in2 := 2)
      I_Contact( #FN_Data.TrackingComponent_2_IsGood )
   END_RUNG wire#w2
   RUNG wire#w1
      { S7_Templates := "SrcType := Int" } GE_Contact(in1 := #IN_Component_Quantity, in2 := 3)
      Contact( #FN_Data.TrackingComponent_3_OnHold )
   END_RUNG wire#w2
   RUNG wire#w1
      { S7_Templates := "SrcType := Int" } GE_Contact(in1 := #IN_Component_Quantity, in2 := 3)
      I_Contact( #FN_Data.TrackingComponent_3_IsGood )
   END_RUNG wire#w2
   RUNG wire#w1
      { S7_Templates := "SrcType := Int" } GE_Contact(in1 := #IN_Component_Quantity, in2 := 4)
      Contact( #FN_Data.TrackingComponent_4_OnHold )
   END_RUNG wire#w2
   RUNG wire#w1
      { S7_Templates := "SrcType := Int" } GE_Contact(in1 := #IN_Component_Quantity, in2 := 4)
      I_Contact( #FN_Data.TrackingComponent_4_IsGood )
   END_RUNG wire#w2
   RUNG wire#w1
      { S7_Templates := "SrcType := Int" } GE_Contact(in1 := #IN_Component_Quantity, in2 := 5)
      Contact( #FN_Data.TrackingComponent_5_OnHold )
   END_RUNG wire#w2
   RUNG wire#w1
      { S7_Templates := "SrcType := Int" } GE_Contact(in1 := #IN_Component_Quantity, in2 := 5)
      I_Contact( #FN_Data.TrackingComponent_5_IsGood )
   END_RUNG wire#w2
   RUNG wire#w1
      { S7_Templates := "SrcType := Int" } GE_Contact(in1 := #IN_Component_Quantity, in2 := 6)
      Contact( #FN_Data.TrackingComponent_6_OnHold )
   END_RUNG wire#w2
   RUNG wire#w1
      { S7_Templates := "SrcType := Int" } GE_Contact(in1 := #IN_Component_Quantity, in2 := 6)
      I_Contact( #FN_Data.TrackingComponent_6_IsGood )
   END_RUNG wire#w2
   RUNG wire#w1
      { S7_Templates := "SrcType := Int" } GE_Contact(in1 := #IN_Component_Quantity, in2 := 7)
      Contact( #FN_Data.TrackingComponent_7_OnHold )
   END_RUNG wire#w2
   RUNG wire#w1
      { S7_Templates := "SrcType := Int" } GE_Contact(in1 := #IN_Component_Quantity, in2 := 7)
      I_Contact( #FN_Data.TrackingComponent_7_IsGood )
   END_RUNG wire#w2
   RUNG wire#w1
      { S7_Templates := "SrcType := Int" } GE_Contact(in1 := #IN_Component_Quantity, in2 := 8)
      Contact( #FN_Data.TrackingComponent_8_OnHold )
   END_RUNG wire#w2
   RUNG wire#w1
      { S7_Templates := "SrcType := Int" } GE_Contact(in1 := #IN_Component_Quantity, in2 := 8)
      I_Contact( #FN_Data.TrackingComponent_8_IsGood )
   END_RUNG wire#w2
   RUNG wire#w1
      { S7_Templates := "SrcType := Int" } GE_Contact(in1 := #IN_Component_Quantity, in2 := 9)
      Contact( #FN_Data.TrackingComponent_9_OnHold )
   END_RUNG wire#w2
   RUNG wire#w1
      { S7_Templates := "SrcType := Int" } GE_Contact(in1 := #IN_Component_Quantity, in2 := 9)
      I_Contact( #FN_Data.TrackingComponent_9_IsGood )
   END_RUNG wire#w2
   RUNG wire#w1
      { S7_Templates := "SrcType := Int" } GE_Contact(in1 := #IN_Component_Quantity, in2 := 10)
      Contact( #FN_Data.TrackingComponent_10_OnHold )
   END_RUNG wire#w2
   RUNG wire#w1
      { S7_Templates := "SrcType := Int" } GE_Contact(in1 := #IN_Component_Quantity, in2 := 10)
      I_Contact( #FN_Data.TrackingComponent_10_IsGood )
   END_RUNG wire#w2
   // the same network as SCL:
   #FN_Data.White_LT_Flash := #FlexNet_DataReceivedByHost AND #IN_OEM_Data.TransactionType.%X3 AND (#FN_Data.ParentPartOnHold OR NOT #FN_Data.ParentPartIsGood OR ((#IN_Component_Quantity >= 1) AND #FN_Data.TrackingComponent_1_OnHold) OR ((#IN_Component_Quantity >= 1) AND NOT #FN_Data.TrackingComponent_1_IsGood) OR ((#IN_Component_Quantity >= 2) AND #FN_Data.TrackingComponent_2_OnHold) OR ((#IN_Component_Quantity >= 2) AND NOT #FN_Data.TrackingComponent_2_IsGood) OR ((#IN_Component_Quantity >= 3) AND #FN_Data.TrackingComponent_3_OnHold) OR ((#IN_Component_Quantity >= 3) AND NOT #FN_Data.TrackingComponent_3_IsGood) OR ((#IN_Component_Quantity >= 4) AND #FN_Data.TrackingComponent_4_OnHold) OR ((#IN_Component_Quantity >= 4) AND NOT #FN_Data.TrackingComponent_4_IsGood) OR ((#IN_Component_Quantity >= 5) AND #FN_Data.TrackingComponent_5_OnHold) OR ((#IN_Component_Quantity >= 5) AND NOT #FN_Data.TrackingComponent_5_IsGood) OR ((#IN_Component_Quantity >= 6) AND #FN_Data.TrackingComponent_6_OnHold) OR ((#IN_Component_Quantity >= 6) AND NOT #FN_Data.TrackingComponent_6_IsGood) OR ((#IN_Component_Quantity >= 7) AND #FN_Data.TrackingComponent_7_OnHold) OR ((#IN_Component_Quantity >= 7) AND NOT #FN_Data.TrackingComponent_7_IsGood) OR ((#IN_Component_Quantity >= 8) AND #FN_Data.TrackingComponent_8_OnHold) OR ((#IN_Component_Quantity >= 8) AND NOT #FN_Data.TrackingComponent_8_IsGood) OR ((#IN_Component_Quantity >= 9) AND #FN_Data.TrackingComponent_9_OnHold) OR ((#IN_Component_Quantity >= 9) AND NOT #FN_Data.TrackingComponent_9_IsGood) OR ((#IN_Component_Quantity >= 10) AND #FN_Data.TrackingComponent_10_OnHold) OR ((#IN_Component_Quantity >= 10) AND NOT #FN_Data.TrackingComponent_10_IsGood));
END_REGION

REGION Network 21: White Light Solid
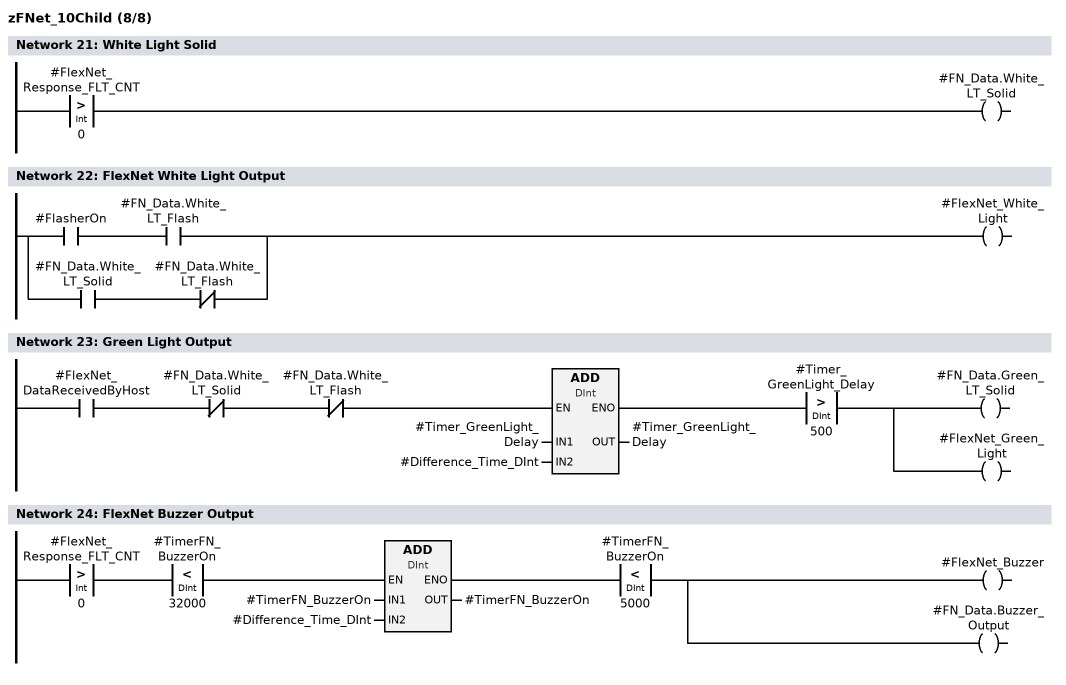
   RUNG wire#powerrail
      { S7_Templates := "SrcType := Int" } GT_Contact(in1 := #FlexNet_Response_FLT_CNT, in2 := 0)
      Coil( #FN_Data.White_LT_Solid )
   END_RUNG
   // the same network as SCL:
   #FN_Data.White_LT_Solid := #FlexNet_Response_FLT_CNT > 0;
END_REGION

REGION Network 22: FlexNet White Light Output
   RUNG wire#powerrail
      Contact( #FlasherOn )
      Contact( #FN_Data.White_LT_Flash )
      wire#w1
      Coil( #FlexNet_White_Light )
   END_RUNG
   RUNG wire#powerrail
      Contact( #FN_Data.White_LT_Solid )
      I_Contact( #FN_Data.White_LT_Flash )
   END_RUNG wire#w1
   // the same network as SCL:
   #FlexNet_White_Light := (#FlasherOn AND #FN_Data.White_LT_Flash) OR (#FN_Data.White_LT_Solid AND NOT #FN_Data.White_LT_Flash);
END_REGION

REGION Network 23: Green Light Output
   RUNG wire#powerrail
      Contact( #FlexNet_DataReceivedByHost )
      I_Contact( #FN_Data.White_LT_Solid )
      I_Contact( #FN_Data.White_LT_Flash )
      { S7_Templates := "SrcType := DInt"; S7_GenerateENO := "TRUE" } Add(in1 := #Timer_GreenLight_Delay, in2 := #Difference_Time_DInt, out => #Timer_GreenLight_Delay)
      { S7_Templates := "SrcType := DInt" } GT_Contact(in1 := #Timer_GreenLight_Delay, in2 := 500)
      wire#w1
      Coil( #FN_Data.Green_LT_Solid )
   END_RUNG
   RUNG wire#w1
      Coil( #FlexNet_Green_Light )
   END_RUNG
   // the same network as SCL:
   // ENO of a box is taken as its EN; it also drops when the box reports an error
   #_w1 := #FlexNet_DataReceivedByHost AND NOT #FN_Data.White_LT_Solid AND NOT #FN_Data.White_LT_Flash;
   IF #_w1 THEN #Timer_GreenLight_Delay := #Timer_GreenLight_Delay + #Difference_Time_DInt; END_IF;
   #FN_Data.Green_LT_Solid := #_w1 AND (#Timer_GreenLight_Delay > 500);
   #FlexNet_Green_Light := #FN_Data.Green_LT_Solid;
END_REGION

REGION Network 24: FlexNet Buzzer Output
   RUNG wire#powerrail
      { S7_Templates := "SrcType := Int" } GT_Contact(in1 := #FlexNet_Response_FLT_CNT, in2 := 0)
      { S7_Templates := "SrcType := DInt" } LT_Contact(in1 := #TimerFN_BuzzerOn, in2 := 32000)
      { S7_Templates := "SrcType := DInt"; S7_GenerateENO := "TRUE" } Add(in1 := #TimerFN_BuzzerOn, in2 := #Difference_Time_DInt, out => #TimerFN_BuzzerOn)
      { S7_Templates := "SrcType := DInt" } LT_Contact(in1 := #TimerFN_BuzzerOn, in2 := 5000)
      wire#w1
      Coil( #FlexNet_Buzzer )
   END_RUNG
   RUNG wire#w1
      Coil( #FN_Data.Buzzer_Output )
   END_RUNG
   // the same network as SCL:
   // ENO of a box is taken as its EN; it also drops when the box reports an error
   #_w1 := (#FlexNet_Response_FLT_CNT > 0) AND (#TimerFN_BuzzerOn < 32000);
   IF #_w1 THEN #TimerFN_BuzzerOn := #TimerFN_BuzzerOn + #Difference_Time_DInt; END_IF;
   #FlexNet_Buzzer := #_w1 AND (#TimerFN_BuzzerOn < 5000);
   #FN_Data.Buzzer_Output := #FlexNet_Buzzer;
END_REGION
END_FUNCTION_BLOCK
